SUBAPPLICATION RegisterMultipleServicesHTTP (* Register many services with different serviceDefinition and serviceURI *)
  (* Standard: 61499-2; Description: Copyright (c) 2019 fortiss GmbH This program and the accompanying materials are made available under the terms of the Eclipse Public License 2.0 which is available at https://www.eclipse.org/legal/epl-2.0/ SPDX-License-Identifier: PL-2.0 *)
  (* Version 1.0, 2019-02-08, Jose Cabral, fortiss GmbH *)
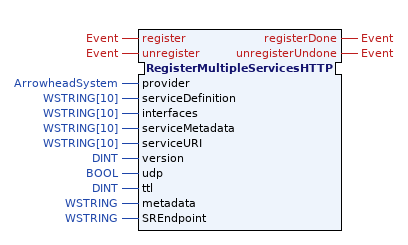
  EVENT_INPUT
    register; (* Register the services *)
    unregister; (* Unregister the services *)
  END_EVENT
  EVENT_OUTPUT
    registerDone; (* Services registered *)
    unregisterUndone; (* Services unregistered *)
  END_EVENT
  VAR_INPUT
    provider : ArrowheadSystem; (* ArrowheadSystem that is providing the Service *)
    serviceDefinition : ARRAY [0..9] OF WSTRING; (* Identifications of the services *)
    interfaces : ARRAY [0..9] OF WSTRING; (* Interfaces implemented by the service *)
    serviceMetadata : ARRAY [0..9] OF WSTRING; (* Metadata of the service in key=value format *)
    serviceURI : ARRAY [0..9] OF WSTRING; (* The URL subpaths of the Services within the address:port of the Provider *)
    version : DINT; (* The version numbering of the Service provided *)
    udp : BOOL; (* True, if the service is provided via UDP. By default, it is false *)
    ttl : DINT; (* Service validity time period expressed in seconds. This gets converted to a date-time, and stored in the database *)
    metadata : WSTRING; (* Metadata belonging to a service/provider pair *)
    SREndpoint : WSTRING; (* Endpoint (IP:PORT/URI) of the Service Registry *)
  END_VAR
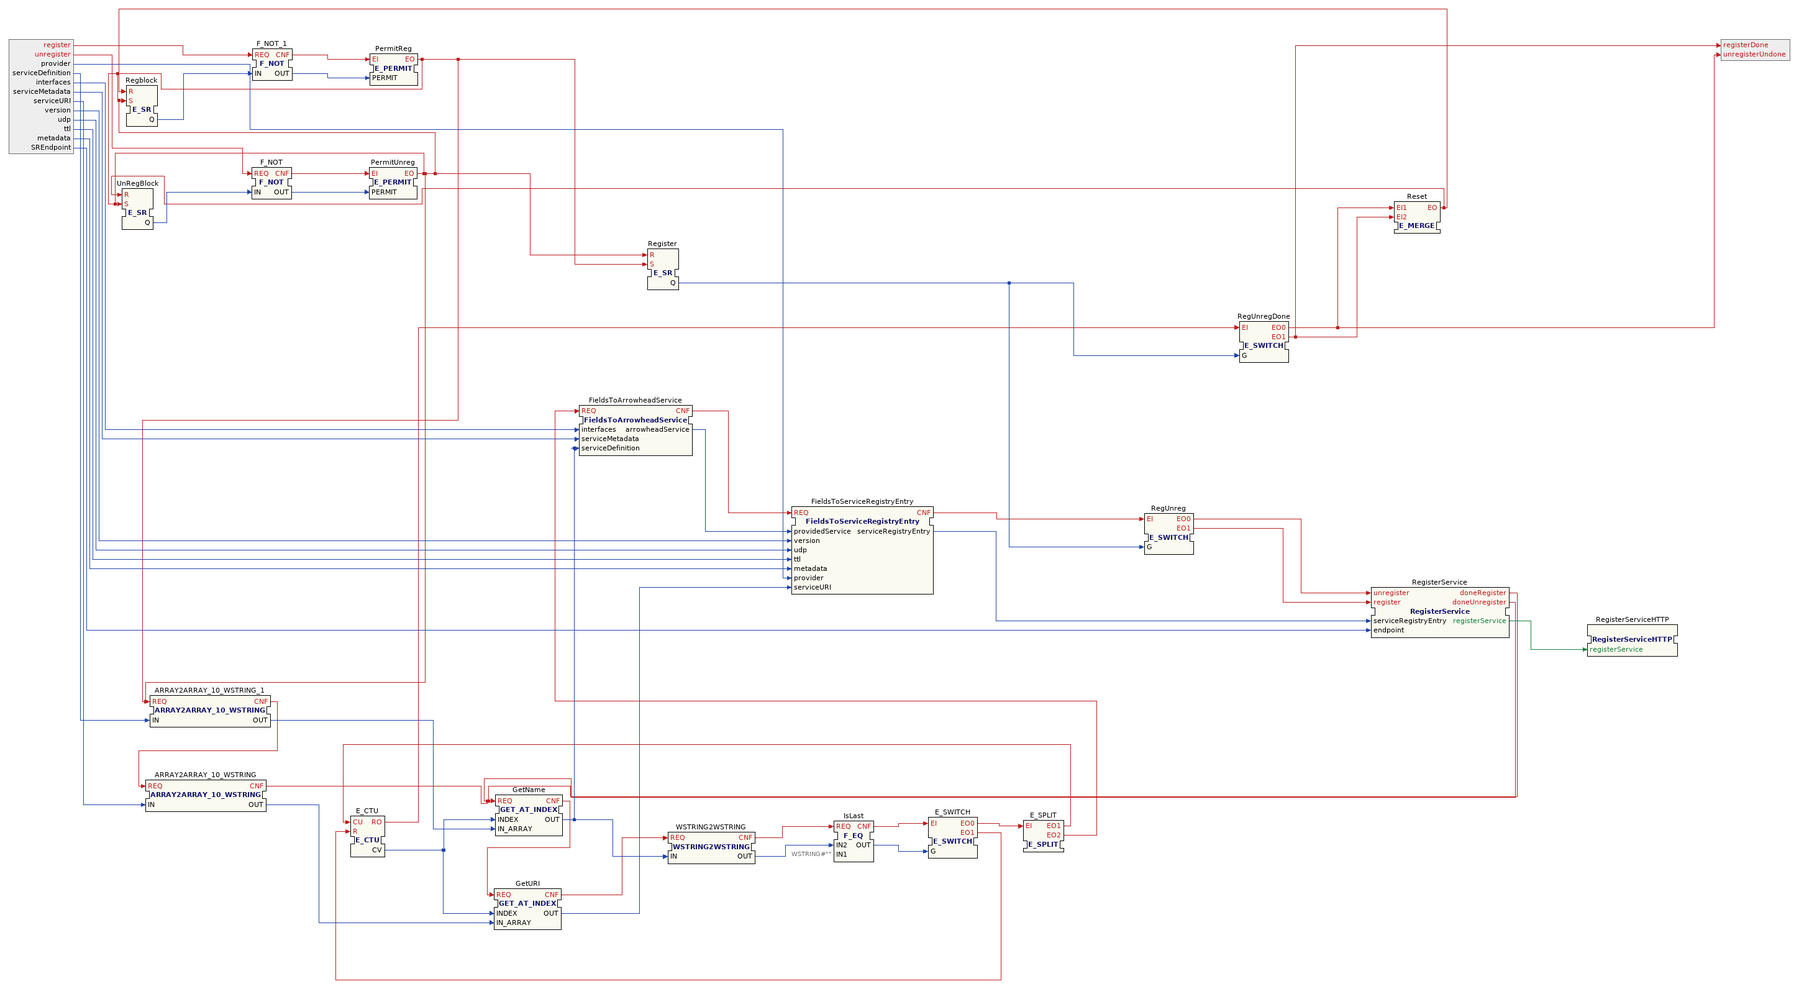
  FBS
    Reset : E_MERGE;
    FieldsToArrowheadService : FieldsToArrowheadService;
    RegUnreg : E_SWITCH;
    Register : E_SR;
    RegisterService : RegisterService;
    RegisterServiceHTTP : RegisterServiceHTTP;
    RegUnregDone : E_SWITCH;
    FieldsToServiceRegistryEntry : FieldsToServiceRegistryEntry;
    GetName : GET_AT_INDEX;
    E_CTU : E_CTU;
    E_SWITCH : E_SWITCH;
    WSTRING2WSTRING : WSTRING2WSTRING;
    IsLast : F_EQ(IN1 := WSTRING#"");
    GetURI : GET_AT_INDEX;
    E_SPLIT : E_SPLIT;
    PermitUnreg : E_PERMIT;
    F_NOT : F_NOT;
    PermitReg : E_PERMIT;
    Regblock : E_SR;
    F_NOT_1 : F_NOT;
    UnRegBlock : E_SR;
    ARRAY2ARRAY_10_WSTRING : ARRAY2ARRAY_10_WSTRING;
    ARRAY2ARRAY_10_WSTRING_1 : ARRAY2ARRAY_10_WSTRING;
  END_FBS
  EVENT_CONNECTIONS
    RegUnregDone.EO0 TO Reset.EI1;
    RegUnregDone.EO1 TO Reset.EI2;
    FieldsToArrowheadService.CNF TO FieldsToServiceRegistryEntry.REQ;
    FieldsToServiceRegistryEntry.CNF TO RegUnreg.EI;
    RegUnreg.EO0 TO RegisterService.unregister;
    RegUnreg.EO1 TO RegisterService.register;
    RegUnregDone.EO1 TO registerDone;
    RegUnregDone.EO0 TO unregisterUndone;
    IsLast.CNF TO E_SWITCH.EI;
    WSTRING2WSTRING.CNF TO IsLast.REQ;
    GetURI.CNF TO WSTRING2WSTRING.REQ;
    E_SPLIT.EO1 TO E_CTU.CU;
    E_SWITCH.EO0 TO E_SPLIT.EI;
    E_SWITCH.EO1 TO E_CTU.R;
    E_SPLIT.EO2 TO FieldsToArrowheadService.REQ;
    RegisterService.doneRegister TO GetName.REQ;
    E_CTU.RO TO RegUnregDone.EI;
    F_NOT_1.CNF TO PermitReg.EI;
    F_NOT.CNF TO PermitUnreg.EI;
    PermitUnreg.EO TO Register.R;
    PermitReg.EO TO Register.S;
    Reset.EO TO UnRegBlock.R;
    Reset.EO TO Regblock.R;
    register TO F_NOT_1.REQ;
    unregister TO F_NOT.REQ;
    PermitUnreg.EO TO UnRegBlock.S;
    PermitUnreg.EO TO Regblock.S;
    PermitReg.EO TO Regblock.S;
    PermitReg.EO TO UnRegBlock.S;
    RegisterService.doneUnregister TO GetName.REQ;
    ARRAY2ARRAY_10_WSTRING.CNF TO GetName.REQ;
    ARRAY2ARRAY_10_WSTRING_1.CNF TO ARRAY2ARRAY_10_WSTRING.REQ;
    PermitReg.EO TO ARRAY2ARRAY_10_WSTRING_1.REQ;
    PermitUnreg.EO TO ARRAY2ARRAY_10_WSTRING_1.REQ;
    GetName.CNF TO GetURI.REQ;
  END_CONNECTIONS
  DATA_CONNECTIONS
    FieldsToArrowheadService.arrowheadService TO FieldsToServiceRegistryEntry.providedService;
    Register.Q TO RegUnreg.G;
    Register.Q TO RegUnregDone.G;
    FieldsToServiceRegistryEntry.serviceRegistryEntry TO RegisterService.serviceRegistryEntry;
    interfaces TO FieldsToArrowheadService.interfaces;
    serviceMetadata TO FieldsToArrowheadService.serviceMetadata;
    version TO FieldsToServiceRegistryEntry.version;
    udp TO FieldsToServiceRegistryEntry.udp;
    ttl TO FieldsToServiceRegistryEntry.ttl;
    metadata TO FieldsToServiceRegistryEntry.metadata;
    SREndpoint TO RegisterService.endpoint;
    provider TO FieldsToServiceRegistryEntry.provider;
    E_CTU.CV TO GetName.INDEX;
    GetName.OUT TO WSTRING2WSTRING.IN;
    E_CTU.CV TO GetURI.INDEX;
    IsLast.OUT TO E_SWITCH.G;
    WSTRING2WSTRING.OUT TO IsLast.IN2;
    GetURI.OUT TO FieldsToServiceRegistryEntry.serviceURI;
    GetName.OUT TO FieldsToArrowheadService.serviceDefinition;
    F_NOT.OUT TO PermitUnreg.PERMIT;
    UnRegBlock.Q TO F_NOT.IN;
    F_NOT_1.OUT TO PermitReg.PERMIT;
    Regblock.Q TO F_NOT_1.IN;
    ARRAY2ARRAY_10_WSTRING.OUT TO GetURI.IN_ARRAY;
    serviceURI TO ARRAY2ARRAY_10_WSTRING.IN;
    ARRAY2ARRAY_10_WSTRING_1.OUT TO GetName.IN_ARRAY;
    serviceDefinition TO ARRAY2ARRAY_10_WSTRING_1.IN;
  END_CONNECTIONS
  ADAPTER_CONNECTIONS
    RegisterService.registerService TO RegisterServiceHTTP.registerService;
  END_CONNECTIONS
END_SUBAPPLICATION
